// TwinCAT 3 PLC project PLC1
// ProgramVersion: 3.1.4023.0
// libraries:
//   Tc2_Standard, * (Beckhoff Automation GmbH)
//   Tc2_System, * (Beckhoff Automation GmbH)
//   Tc3_Module, * (Beckhoff Automation GmbH)
// project tree:
//   / PlcTask.TcTTO
//   POUs/ FB_Object.TcPOU, MAIN.TcPOU
// real-time tasks:
//   TASK PlcTask: cycle T#10ms, priority 20, ADS port 350

CONFIGURATION PLC1
    RESOURCE PLC ON TwinCAT3
        TASK PlcTask(INTERVAL := T#10ms, PRIORITY := 20);
        PROGRAM MAIN WITH PlcTask : MAIN;
    END_RESOURCE
END_CONFIGURATION

// ---- POUs/MAIN.TcPOU
PROGRAM MAIN
VAR	

	{ attribute 'TcHmiSymbol.AddSymbol' }
	fbObject1 : FB_Object;	
	{ attribute 'TcHmiSymbol.AddSymbol' }
	fbObject2 : FB_Object;	
	{ attribute 'TcHmiSymbol.AddSymbol' }
	fbObject3 : FB_Object;	
	{ attribute 'TcHmiSymbol.AddSymbol' }
	fbObject4 : FB_Object;	
	{ attribute 'TcHmiSymbol.AddSymbol' }
	fbObject5 : FB_Object;	
	{ attribute 'TcHmiSymbol.AddSymbol' }
	fbObject6 : FB_Object;	
	
END_VAR

fbObject1(nObjectID:= 1);
fbObject2(nObjectID:= 2);
fbObject3(nObjectID:= 3);
fbObject4(nObjectID:= 4);
fbObject5(nObjectID:= 5);
fbObject6(nObjectID:= 6);

END_PROGRAM

// ---- POUs/FB_Object.TcPOU
FUNCTION_BLOCK FB_Object
VAR_INPUT
	nObjectID : INT;
END_VAR
VAR
	bActive : BOOL;
	fValue : REAL;
	fbRandom : DRAND;
END_VAR

IF bActive THEN
	fbRandom(Seed:= nObjectID, NUm=> fValue);
END_IF

END_FUNCTION_BLOCK
